// LS Electric XG5000 project: 과년66_3_4
// PLC NewPLC
// module base 0 slot 0: 입출력 모듈:XBC-DR20S (DC 24V 입력 12점, 릴레이 출력 8점)

PROGRAM NewProgram (task: 스캔 프로그램)

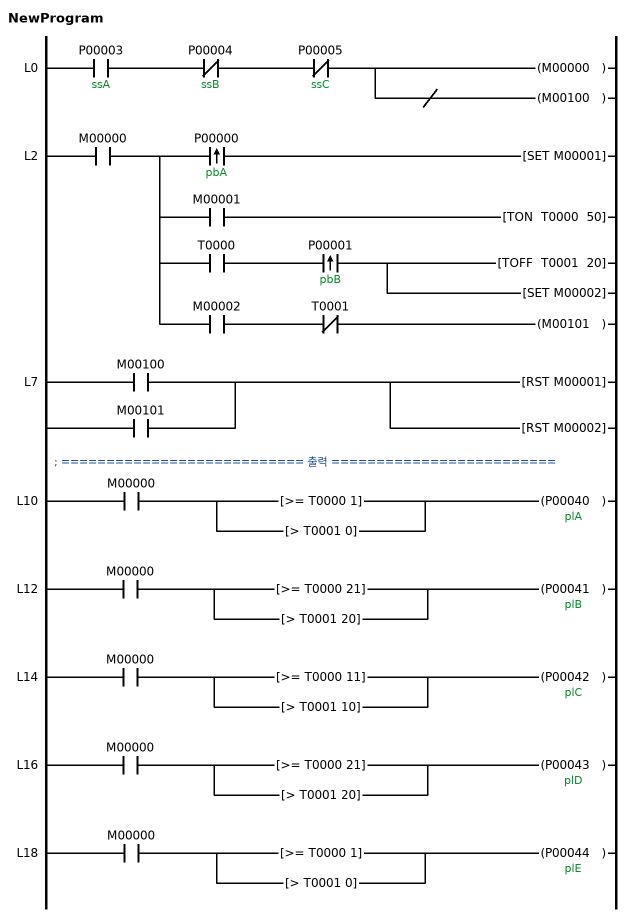
; L0
LOAD      P00003	// ssA
AND NOT   P00004	// ssB
AND NOT   P00005	// ssC
OUT       M00000
NOT
OUT       M00100
; L2
LOAD      M00000
MPUSH
ANDP      P00000	// pbA
SET       M00001
MLOAD
AND       M00001
TON       T0000 50
MLOAD
AND       T0000
ANDP      P00001	// pbB
TOFF      T0001 20
SET       M00002
MPOP
AND       M00002
AND NOT   T0001
OUT       M00101
; L7
LOAD      M00100
OR        M00101
RST       M00001
RST       M00002
// =========================== 출력 =========================
; L10
LOAD      M00000
LOAD>=    T0000 1
OR>       T0001 0
AND LOAD
OUT       P00040	// plA
; L12
LOAD      M00000
LOAD>=    T0000 21
OR>       T0001 20
AND LOAD
OUT       P00041	// plB
; L14
LOAD      M00000
LOAD>=    T0000 11
OR>       T0001 10
AND LOAD
OUT       P00042	// plC
; L16
LOAD      M00000
LOAD>=    T0000 21
OR>       T0001 20
AND LOAD
OUT       P00043	// plD
; L18
LOAD      M00000
LOAD>=    T0000 1
OR>       T0001 0
AND LOAD
OUT       P00044	// plE

VARIABLES AND COMMENTS (devices not used above)
P00002	BIT	pbC